Fanuc KAREL source: kt00365.KL

-- PROVISIONAL review KL for V1013-1; original PC SHA256 85e44d157c06311dea101e81ac120ba78e38d18f644fe041258fdd2ff35420f5
-- Incomplete behavior may be omitted. Consult companion uncertainty JSON. Do not deploy.
PROGRAM KT00365
%NOLOCKGROUP
VAR
  I1 : INTEGER
  I2 : INTEGER
  OUT : BOOLEAN
BEGIN
  -- UNRESOLVED_PC offsets 5-16; opcodes 2E,23
  -- UNRESOLVED_PC offsets 21-32; opcodes 2E,23
  -- UNRESOLVED_PC offsets 37-48; opcodes 2E,23
  -- UNRESOLVED_PC offsets 53-64; opcodes 2E,23
  -- UNRESOLVED_PC offsets 69-88; opcodes 21,21,5A,23
  -- UNRESOLVED_PC offsets 93-97; opcodes 7F
END KT00365
